{attribute 'linkalways'} 
{attribute 'no_explicit_call' := 'This FB is a CLASS and must be accessed using methods or properties'}
{attribute 'enable_dynamic_creation'}
FUNCTION_BLOCK Node_F_VN_MedianElementElementwise_TcVnPoint3_LREAL EXTENDS VisionNode
VAR
    ipContainer : _ITcVnContainer;
    aMedian : _TcVnPoint3_LREAL;
    hrPrev : _HRESULT(S_OK);
    hresult : _HRESULT(S_OK);
END_VAR

METHOD PUBLIC  Clone : I_Node
VAR
	pNode : POINTER TO Node_F_VN_MedianElementElementwise_TcVnPoint3_LREAL;
END_VAR
pNode := __NEW(Node_F_VN_MedianElementElementwise_TcVnPoint3_LREAL);
Clone := pNode^;
END_METHOD

METHOD FB_init : BOOL
VAR_INPUT
	bInitRetains : BOOL; // if TRUE, the retain variables are initialized (warm start / cold start)
	bInCopyCode : BOOL;  // if TRUE, the instance afterwards gets moved into the copy code (online change)
END_VAR
AddInput('ipContainer', ipContainer);
AddInput('aMedian', aMedian);
AddInput('hrPrev', hrPrev);
AddOutput('ipContainer', ipContainer);
AddOutput('hresult',hresult);
END_METHOD

METHOD PROTECTED OnExecute : HRESULT
hresult.Value := F_VN_MedianElementElementwise_TcVnPoint3_LREAL(
    ipContainer := ipContainer.Value,
    aMedian := aMedian.Value,
    hrPrev:= hrPrev.Value);
END_METHOD

METHOD PUBLIC PreExecutionCheck
VAR_INPUT
	Check : I_PreExecutionChecks;
END_VAR
Check.IsTrue(ipContainer.IsValid, 'ipContainer must be a valid container');
END_METHOD

END_FUNCTION_BLOCK

(* stored: Version 1.1.0.1, ProductVersion 3.1.4024.13
   POU Node_F_VN_MedianElementElementwise_TcVnPoint3_LREAL: Id {88bb9056-83bf-40a6-860e-032399711047}, SpecialFunc None
   Folder Constructor: Id {0fbb15c9-042a-49ce-9143-22733bdca1d1}
   Method Clone: Id {86725af2-3306-40fd-8c3c-1329fa140d12}
   Method FB_init: Id {ec7967ef-988b-4c82-9ba6-43a3d9cd6bdf}
   Method OnExecute: Id {6c62c33c-2b02-42a6-9fb5-06ad4bd01d85}
   Method PreExecutionCheck: Id {515fe1e1-b9ac-4c87-8cb1-1999e37b3f1f} *)
